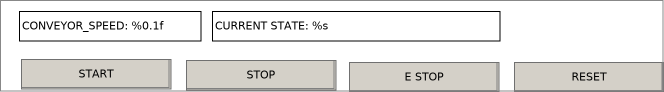
VISUALIZATION Visualization  // 664x92
    Button (21,59 150x30), "START", colour toggle: MAIN.START
        OnMouseDown: toggle MAIN.START
    Button (186,60 150x30), "STOP", colour toggle: MAIN.STOP
        OnMouseDown: toggle MAIN.STOP
    Button (349,62 150x30), "E STOP", colour toggle: MAIN.E_STOP
        OnMouseDown: toggle MAIN.E_STOP
    Button (514,62 150x30), "RESET", colour toggle: MAIN.RESET
        OnMouseDown: toggle MAIN.RESET
    Rectangle (19,11 182x30), "CONVEYOR_SPEED: %0.1f", text variable: MAIN.CONVEYOR_SPEED
    Rectangle (212,11 288x30), "CURRENT STATE: %s", text variable: MAIN.STATE_DISP_STR
END_VISUALIZATION

(* stored: Version 1.1.0.1, ProductVersion 3.1.4024.13
   Visu Visualization: Id {48adab8b-06d5-4030-82fa-b04a66f12c78} *)
